TYPE ST_Motorparam :
STRUCT
	rMaxSpeed		:REAL		:= 2000;//rpm
	rMinSpeed		:REAL		:= 0;	//rpm
END_STRUCT
END_TYPE

(* stored: Version 1.1.0.1, ProductVersion 3.1.4024.12
   DUT ST_Motorparam: Id {492daac1-64e6-47c3-a87b-631d6bad19c8} *)
